FUNCTION_BLOCK FB_Motion_Control
VAR_INPUT
	eStatus : E_Status := E_Status.Checking;
END_VAR
VAR_OUTPUT
	bAutoEnable 							: BOOL;
	bManualEnable 							: BOOL; 
	bSecondaryAutoEnable 					: BOOL; 
	bSecondaryManualEnable				    : BOOL; 

END_VAR
VAR
	fbEncoderScaling 						: FB_EncoderScaling;
	fbAutoStartPos							: FB_AutoStartPos;
	fbAutoSineMotion    					: FB_AutoSineMotion; 
	fbClock_MOOG							: FB_Clock;
	fbClock_dis								: FB_Clock;
	fbDisplacementControl  					: FB_DisplacementControl;
	fbSecondaryControlStartPos				: FB_SecondaryControlStartPos;
	fbJoystick 								: FB_Joystick; 
	fbGetStartPos 							: FB_StartPos;
	fbWinchVelIntegrator					: FB_Integrator;  
	bStartPosOK								: BOOL;
	fWinchVelRefManual						: LREAL; 
	fWinchVelRefAuto                        : LREAL; 
	fWinchPosRefManual						: LREAL; 
	fInitialWinchPos						: LREAL; 
	fbPIDController							: FB_PID_controller_old; 
	
	
	//Secondary control
	
	fbPID 									: FB_PID_controller_old;
	fbFeedForward							: FB_FeedForward;
	
	I_output								: LREAL;
	D_output								: LREAL;
END_VAR
VAR // added by the converter: edge detectors and wires of the graphical bodies
    _w1, _w2 : LREAL;
END_VAR

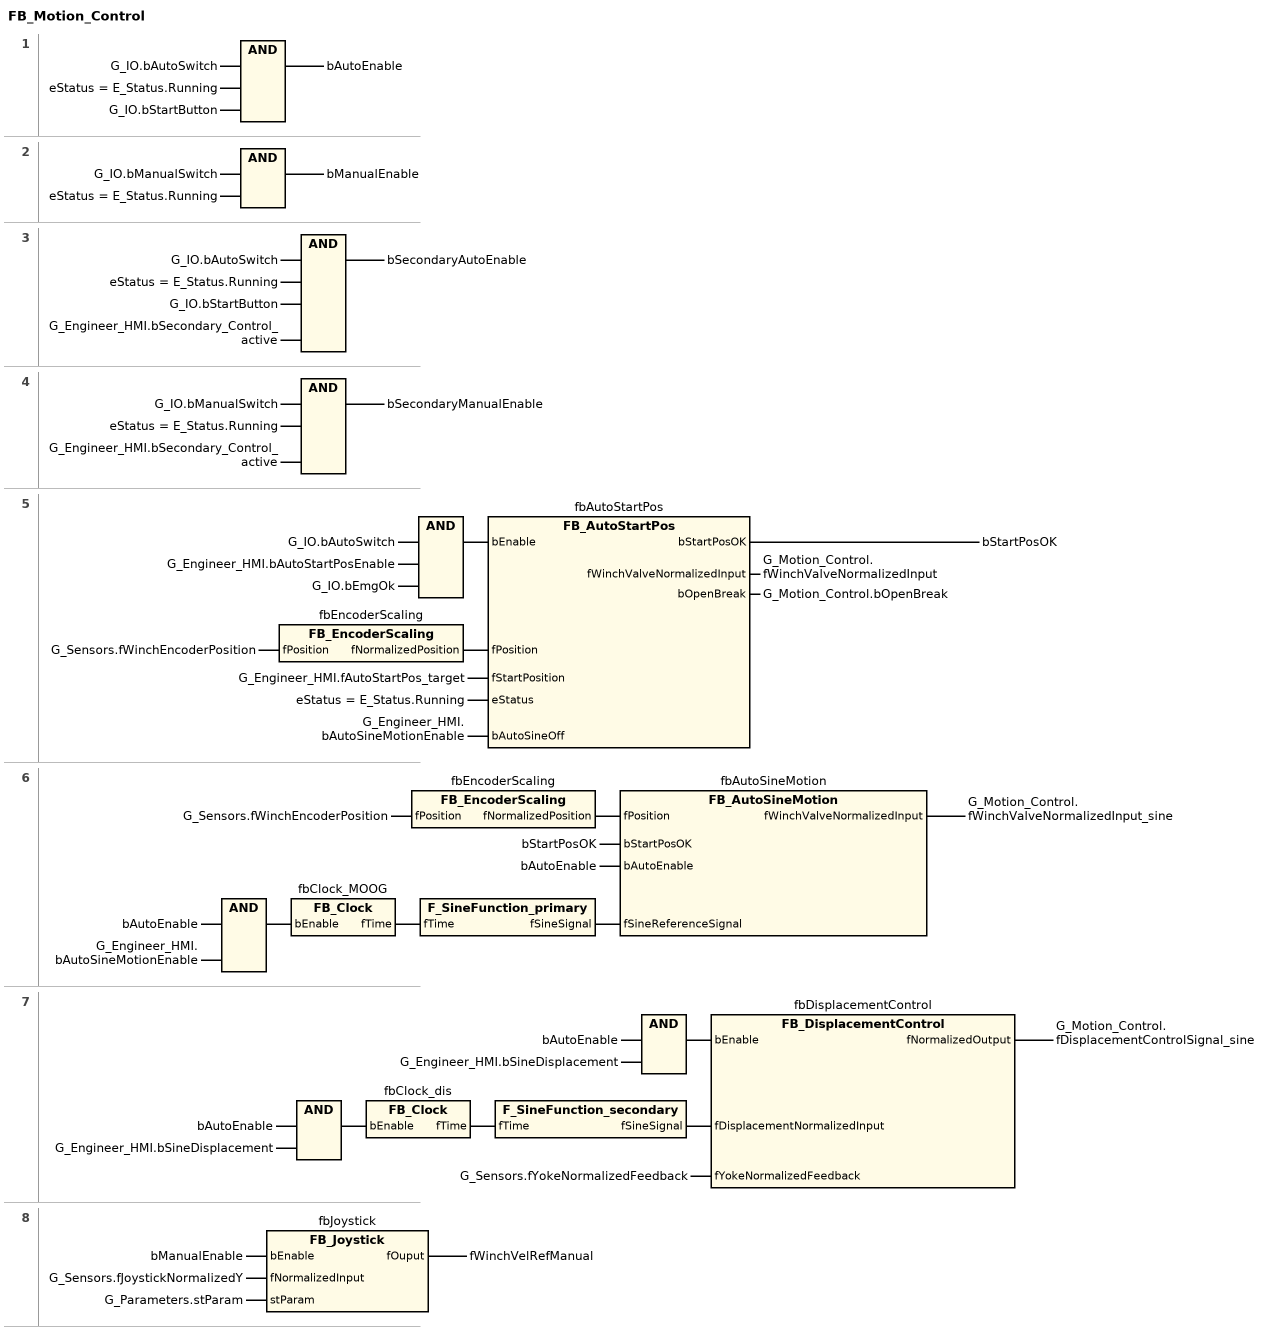
// NETWORK 1
bAutoEnable := G_IO.bAutoSwitch AND (eStatus = E_Status.Running) AND G_IO.bStartButton;

// NETWORK 2
bManualEnable := G_IO.bManualSwitch AND (eStatus = E_Status.Running);

// NETWORK 3
bSecondaryAutoEnable := G_IO.bAutoSwitch AND (eStatus = E_Status.Running) AND G_IO.bStartButton AND G_Engineer_HMI.bSecondary_Control_active;

// NETWORK 4
bSecondaryManualEnable := G_IO.bManualSwitch AND (eStatus = E_Status.Running) AND G_Engineer_HMI.bSecondary_Control_active;

// NETWORK 5
fbEncoderScaling(fPosition := G_Sensors.fWinchEncoderPosition); // FB_EncoderScaling
fbAutoStartPos(
    bEnable := G_IO.bAutoSwitch AND G_Engineer_HMI.bAutoStartPosEnable AND G_IO.bEmgOk,
    fPosition := fbEncoderScaling.fNormalizedPosition,
    fStartPosition := G_Engineer_HMI.fAutoStartPos_target,
    eStatus := eStatus = E_Status.Running,
    bAutoSineOff := G_Engineer_HMI.bAutoSineMotionEnable,
    fWinchValveNormalizedInput => G_Motion_Control.fWinchValveNormalizedInput,
    bOpenBreak => G_Motion_Control.bOpenBreak); // FB_AutoStartPos
bStartPosOK := fbAutoStartPos.bStartPosOK;

// NETWORK 6
fbEncoderScaling(fPosition := G_Sensors.fWinchEncoderPosition); // FB_EncoderScaling
fbClock_MOOG(bEnable := bAutoEnable AND G_Engineer_HMI.bAutoSineMotionEnable); // FB_Clock
F_SineFunction_primary(fTime := fbClock_MOOG.fTime, fSineSignal => _w1);
fbAutoSineMotion(
    fPosition := fbEncoderScaling.fNormalizedPosition,
    bStartPosOK := bStartPosOK,
    bAutoEnable := bAutoEnable,
    fSineReferenceSignal := _w1); // FB_AutoSineMotion
G_Motion_Control.fWinchValveNormalizedInput_sine := fbAutoSineMotion.fWinchValveNormalizedInput;

// NETWORK 7
fbClock_dis(bEnable := bAutoEnable AND G_Engineer_HMI.bSineDisplacement); // FB_Clock
F_SineFunction_secondary(fTime := fbClock_dis.fTime, fSineSignal => _w2);
fbDisplacementControl(
    bEnable := bAutoEnable AND G_Engineer_HMI.bSineDisplacement,
    fDisplacementNormalizedInput := _w2,
    fYokeNormalizedFeedback := G_Sensors.fYokeNormalizedFeedback); // FB_DisplacementControl
G_Motion_Control.fDisplacementControlSignal_sine := fbDisplacementControl.fNormalizedOutput;

// NETWORK 8
fbJoystick(
    bEnable := bManualEnable,
    fNormalizedInput := G_Sensors.fJoystickNormalizedY,
    stParam := G_Parameters.stParam); // FB_Joystick
fWinchVelRefManual := fbJoystick.fOuput;

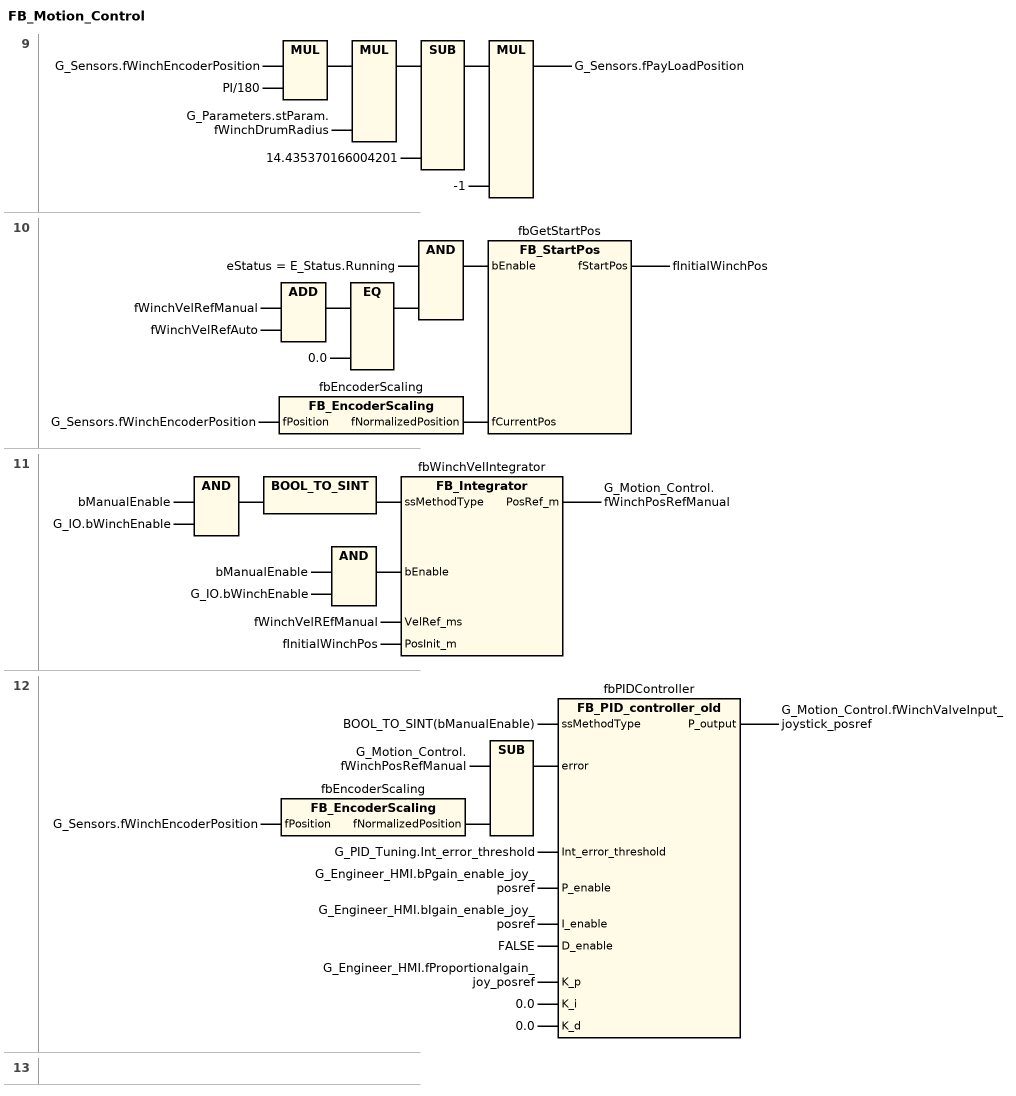
// NETWORK 9
G_Sensors.fPayLoadPosition := ((G_Sensors.fWinchEncoderPosition * (PI/180)) * G_Parameters.stParam.fWinchDrumRadius - 14.435370166004201) * -1;

// NETWORK 10
fbEncoderScaling(fPosition := G_Sensors.fWinchEncoderPosition); // FB_EncoderScaling
fbGetStartPos(bEnable := (eStatus = E_Status.Running) AND fWinchVelRefManual + fWinchVelRefAuto = 0.0, fCurrentPos := fbEncoderScaling.fNormalizedPosition); // FB_StartPos
fInitialWinchPos := fbGetStartPos.fStartPos;

// NETWORK 11
fbWinchVelIntegrator(
    ssMethodType := BOOL_TO_SINT(bManualEnable AND G_IO.bWinchEnable),
    bEnable := bManualEnable AND G_IO.bWinchEnable,
    VelRef_ms := fWinchVelREfManual,
    PosInit_m := fInitialWinchPos); // FB_Integrator
G_Motion_Control.fWinchPosRefManual := fbWinchVelIntegrator.PosRef_m;

// NETWORK 12
fbEncoderScaling(fPosition := G_Sensors.fWinchEncoderPosition); // FB_EncoderScaling
fbPIDController(
    ssMethodType := BOOL_TO_SINT(bManualEnable),
    error := G_Motion_Control.fWinchPosRefManual - fbEncoderScaling.fNormalizedPosition,
    Int_error_threshold := G_PID_Tuning.Int_error_threshold,
    P_enable := G_Engineer_HMI.bPgain_enable_joy_posref,
    I_enable := G_Engineer_HMI.bIgain_enable_joy_posref,
    D_enable := FALSE,
    K_p := G_Engineer_HMI.fProportionalgain_joy_posref,
    K_i := 0.0,
    K_d := 0.0); // FB_PID_controller_old
G_Motion_Control.fWinchValveInput_joystick_posref := fbPIDController.P_output;

// NETWORK 13

END_FUNCTION_BLOCK

(* stored: Version 1.1.0.1
   POU FB_Motion_Control: Id {b91e27fc-a1b6-46fc-99a4-88a21e344525}, SpecialFunc None *)
